TYPE U_ReceivedData :
UNION
	DataArray	: ARRAY[0 .. 255] OF BYTE;
	DataString	: STRING(255);
END_UNION
END_TYPE

(* stored: Version 1.1.0.1, ProductVersion 3.1.4024.13
   DUT U_ReceivedData: Id {d8a6f817-9a8f-4e7b-a29a-658129e1b2a9} *)
